{attribute 'TcGenerated'}
// This function has been automatically generated from the project information.
VAR_GLOBAL CONSTANT
	{attribute 'const_non_replaced'}
	{attribute 'linkalways'}
	stLibVersion_MyLibrary01 : ST_LibVersion := (iMajor := 2, iMinor := 0, iBuild := 0, iRevision := 0, sVersion := '2.0.0.0');
END_VAR

(* stored: Version 1.1.0.1, ProductVersion 3.1.4020.6
   GVL Global_Version: Id {003ddff5-6a56-467e-b69a-0798fad84940} *)
